TYPE SampleDataStructure : 
STRUCT
    SampleString : STRING;
    SampleString2 : STRING := '3retewtertert2342345*-+/';
    SampleInt : INT;
    SampleInt2 : INT := 432;
    SampleBool : BOOL;
    SampleBool2 : BOOL := TRUE;
    SampleWString : WSTRING;
    SampleLREAL : LREAL;
    SampleNestedStructure : SampleDataStructureLevel2;
END_STRUCT
END_TYPE

(* stored: Version 1.1.0.1, ProductVersion 3.1.4024.9
   DUT SampleDataStructure: Id {0e62a0f6-a025-0f0f-3eb3-7f26678fac54} *)
